{attribute 'qualified_only'}
VAR_GLOBAL CONSTANT
	
END_VAR
VAR_GLOBAL CONSTANT
	PI_2_MIL: DINT := 6283185;
	COUNT: DINT := 1048576;
END_VAR

(* stored: Version 1.1.0.1, ProductVersion 3.1.4024.11
   GVL CONST: Id {92f96cdf-9708-43bf-a5f1-4276328fdb5c}, ParameterList True *)
